(*
ST_Safety does not point directly to the raw EtherCAT data. Instead,
mLinkRefs() links ST_Safety reference members to this structure.
*)
TYPE ST_PNOZEtherCATIn :
STRUCT
    aSafetyFunctionIn: ARRAY[GVL_SafetyIO.cLOWER_BOUND_SF..GVL_SafetyIO.cUPPER_BOUND_SF] OF ST_SafetyFunctionIn; //Input Byte 04..11
    stLEDState: ST_LEDState; //Input Byte 16

    stTableNumberIn: ST_TableNumberIn; //Input Byte 17
    stSegmentNumberIn: ST_SegmentNumberIn; //Input Byte 18

    stSafetyStatus: ST_SafetyStatus; //Placeholder, WIP
    aSubSystemIn: ARRAY[1..GVL_SafetyIO.cUPPER_NBR_OF_SS] OF ST_SubSystemIn; //Placeholder, WIP
    stSequenceIn: ST_SequenceIn; //Placeholder, WIP
END_STRUCT
END_TYPE

(* stored: Version 1.1.0.1
   DUT ST_PNOZEtherCATIn: Id {4d26afb5-ffd0-0d85-0f77-77acb686f585} *)
